DATA_BLOCK DB 17
TITLE =
{ S7_language := '7(1) Deutsch (Deutschland)  10.06.2014  10:57:37' }
AUTHOR : DAGO
FAMILY : PEPS
NAME : PEPS
VERSION : 0.1


  STRUCT
   alarms : STRUCT
    alarms : ARRAY  [1 .. 50 ] OF WORD;
   END_STRUCT ;
   LOT_DATA : STRUCT
    SON : STRING  [10 ];
    INR : STRING  [15 ];
    LOTSIZE : DINT ;
    SPARE_34 : DWORD ;
    SPARE_38 : DWORD ;
    SPARE_42 : DWORD ;
    SPARE_46 : DWORD ;
   END_STRUCT ;
   GENERAL : STRUCT
    MODE : INT ;
    RFD : BOOL ;
    RFU : BOOL ;
    RUN : BOOL ;
    IDLE : BOOL ;
    SPARE_2_4 : BOOL ;
    SPARE_2_5 : BOOL ;
    SPARE_2_6 : BOOL ;
    SPARE_2_7 : BOOL ;
    MACHINE_STARTED : BOOL ;	//Machine started
    AUTO : BOOL ;	//Auto visualisation
    MANUAL : BOOL ;	//Manual visualisation
    STELLEN : BOOL ;	//Stellen
    INFEED_BLOCKING : BOOL ;	//Infeed blocking visualisation
    PRODUCT_SUPPLY : BOOL ;	//Product supply visualisation
    PRE_PRODUCTION : BOOL ;	//Pr� production visualisation
    FILLING : BOOL ;	//Filling visualisation
    STOPPERS : BOOL  := TRUE;	//Stoppers visualisation
    IPC_SAMPLING : BOOL ;	//IPC sampling visualisation
    REJECT_ALL_SYRINGES : BOOL ;	//Reject all syringes visualisation
    RUN_EMPTY : BOOL ;	//Run empty machine visualisation
    START_UP : BOOL ;	//StartUp visualisation
    PRIMING : BOOL ;	//Priming visualisation
    PREPRODUCTION : BOOL ;	//Pr� production visualisation
    RECIRCULATION_DEACTIVE : BOOL ;	//Recirculation deactivated
    SPARE_5_0 : BOOL ;
    SPARE_5_1 : BOOL ;
    SPARE_5_2 : BOOL ;
    SPARE_5_3 : BOOL ;
    SPARE_5_4 : BOOL ;
    SPARE_5_5 : BOOL ;
    SPARE_5_6 : BOOL ;
    SPARE_5_7 : BOOL ;
    SPARE_6_0 : BOOL ;
    SPARE_6_1 : BOOL ;
    SPARE_6_2 : BOOL ;
    SPARE_6_3 : BOOL ;
    SPARE_6_4 : BOOL ;
    SPARE_6_5 : BOOL ;
    SPARE_6_6 : BOOL ;
    SPARE_6_7 : BOOL ;
    PHASE : INT ;	//Phase
    SUB_PHASE : INT ;	//Sub Phase
    SPARE_12 : INT ;
    SPARE_14 : INT ;
    SPARE_16 : INT ;
    SPARE_18 : INT ;
    SPARE_20 : INT ;
    SPARE_22 : INT ;
    SPARE_24 : INT ;
    SPARE_26 : INT ;
    SPARE_28 : INT ;
    SPARE_30 : INT ;
    SPARE_32 : INT ;
    SPARE_34 : INT ;
    SPARE_36 : INT ;
    SPARE_38 : INT ;
    SPARE_40 : INT ;
    SPARE_42 : INT ;
    SPARE_44 : INT ;
    SPARE_46 : INT ;
    SPARE_48 : WORD ;
   END_STRUCT ;
   COUNTERS : STRUCT
    TOTAL_GOOD : DINT ;	//Aantal goede stuks
    REJECT_FILLER_CAPPER : DINT ;	//Aantal uitgeworpen
    REJECT_PRIMING : INT ;	//Aantal gebruikt voor priming
    TOTAL_OBJECTS : DINT ;	//Totaal aantal
    FILLED_REJECTED : DINT ;	//Aantal gevuld en uitgeworpen
    NON_FILLED_REJECTED : DINT ;	//Aantal niet gevuld en uitgeworpen
    IPC_FILLED_SAMPLES : INT ;	//Aantal als staal genomen
    REJECT_NON_STARTUP : DINT ;	//Aantal fouten door geen opstart, priming of pr�-produktie uit te voeren
    SPARE_28 : INT ;
    REJECT_NEEDLE_DOWN : INT ;	//Aantal uitgeworpen na naalden uit positie
    REJECT_ALL_NON_FILL_SYR : DINT ;	//Aantal niet gevulde uitgeworpen door functie 'Alle syringes uitwerpen'
    REJECT_ALL_FILLED_SYR : DINT ;	//Aantal gevulde uitgeworpen door functie 'Alle syringes uitwerpen'
    FAULT_TIP_CAP_CONTR : INT ;	//Aantal fouten aan tip cap controlestation
    FAULT_TIP_CAP_CONTR_1 : INT ;	//Aantal fouten aan tip cap controle positie 1
    FAULT_TIP_CAP_CONTR_2 : INT ;	//Aantal fouten aan tip cap controle positie 2
    FAULT_TIP_CAP_CONTR_3 : INT ;	//Aantal fouten aan tip cap controle positie 3
    FAULT_TIP_CAP_CONTR_4 : INT ;	//Aantal fouten aan tip cap controle positie 4
    FAULT_STOPPER_CONTR : INT ;	//Aantal fouten aan stopper controlestation
    FAULT_STOPPER_CONTR_1 : INT ;	//Aantal fouten aan stopper controle positie 1
    FAULT_STOPPER_CONTR_2 : INT ;	//Aantal fouten aan stopper controle positie 2
    FAULT_STOPPER_CONTR_3 : INT ;	//Aantal fouten aan stopper controle positie 3
    FAULT_STOPPER_CONTR_4 : INT ;	//Aantal fouten aan stopper controle positie 4
    FAULT_STANDSTILL : DINT ;	//Aantal slecht door maximale stilstand overschreden
    FAULT_TUNNEL : DINT ;	//Aantal slecht door te lang in tunnel
    FAULT_ISOL_FILLED : DINT ;	//Aantal gevulde slecht door isolator
    FAULT_ISOL_NON_FILLED : DINT ;	//Aantal niet gevulde slecht door isolator
    FAULT_E_STOP_FILLED : DINT ;	//Aantal slechten onder vulnaalden door activatie noodstop
    FAULT_E_STOP_NON_FILLED : DINT ;	//Aantal slechten tussen vullen en stopperen door activatie noodstop
    REJECT_SMC_MODE : DINT ;	//Aantal uitgeworpen in SMC mode
    REJECT_JOG_MODE : DINT ;	//Aantal uitgeworpen in JOG mode
    SPARE_92 : DINT ;
    REJECT_RECIRCULATION : DINT ;	//Aantal uitgeworpen na recirculatie
    SPARE_100 : DINT ;
    SPARE_104 : DINT ;
    SPARE_108 : DINT ;
    SPARE_112 : DINT ;
    SPARE_116 : DINT ;
    SPARE_120 : DINT ;
    SPARE_124 : DINT ;
    SPARE_128 : INT ;
   END_STRUCT ;
   SPARE_288 : DWORD ;
   SPARE_292 : DWORD ;
   SPARE_296 : DWORD ;
   SPARE_290 : DWORD ;
   SPARE_294 : DWORD ;
  END_STRUCT ;
BEGIN
   ALARMS.ALARM[1] := FALSE;
   ALARMS.ALARM[2] := FALSE;
   ALARMS.ALARM[3] := FALSE;
   ALARMS.ALARM[4] := FALSE;
   ALARMS.ALARM[5] := FALSE;
   ALARMS.ALARM[6] := FALSE;
   ALARMS.ALARM[7] := FALSE;
   ALARMS.ALARM[8] := FALSE;
   ALARMS.ALARM[9] := FALSE;
   ALARMS.ALARM[10] := FALSE;
   ALARMS.ALARM[11] := FALSE;
   ALARMS.ALARM[12] := FALSE;
   ALARMS.ALARM[13] := FALSE;
   ALARMS.ALARM[14] := FALSE;
   ALARMS.ALARM[15] := FALSE;
   ALARMS.ALARM[16] := FALSE;
   ALARMS.ALARM[17] := FALSE;
   ALARMS.ALARM[18] := FALSE;
   ALARMS.ALARM[19] := FALSE;
   ALARMS.ALARM[20] := FALSE;
   ALARMS.ALARM[21] := FALSE;
   ALARMS.ALARM[22] := FALSE;
   ALARMS.ALARM[23] := FALSE;
   ALARMS.ALARM[24] := FALSE;
   ALARMS.ALARM[25] := FALSE;
   ALARMS.ALARM[26] := FALSE;
   ALARMS.ALARM[27] := FALSE;
   ALARMS.ALARM[28] := FALSE;
   ALARMS.ALARM[29] := FALSE;
   ALARMS.ALARM[30] := FALSE;
   ALARMS.ALARM[31] := FALSE;
   ALARMS.ALARM[32] := FALSE;
   ALARMS.ALARM[33] := FALSE;
   ALARMS.ALARM[34] := FALSE;
   ALARMS.ALARM[35] := FALSE;
   ALARMS.ALARM[36] := FALSE;
   ALARMS.ALARM[37] := FALSE;
   ALARMS.ALARM[38] := FALSE;
   ALARMS.ALARM[39] := FALSE;
   ALARMS.ALARM[40] := FALSE;
   ALARMS.ALARM[41] := FALSE;
   ALARMS.ALARM[42] := FALSE;
   ALARMS.ALARM[43] := FALSE;
   ALARMS.ALARM[44] := FALSE;
   ALARMS.ALARM[45] := FALSE;
   ALARMS.ALARM[46] := FALSE;
   ALARMS.ALARM[47] := FALSE;
   ALARMS.ALARM[48] := FALSE;
   ALARMS.ALARM[49] := FALSE;
   ALARMS.ALARM[50] := FALSE;
   ALARMS.ALARM[51] := FALSE;
   ALARMS.ALARM[52] := FALSE;
   ALARMS.ALARM[53] := FALSE;
   ALARMS.ALARM[54] := FALSE;
   ALARMS.ALARM[55] := FALSE;
   ALARMS.ALARM[56] := FALSE;
   ALARMS.ALARM[57] := FALSE;
   ALARMS.ALARM[58] := FALSE;
   ALARMS.ALARM[59] := FALSE;
   ALARMS.ALARM[60] := FALSE;
   ALARMS.ALARM[61] := FALSE;
   ALARMS.ALARM[62] := FALSE;
   ALARMS.ALARM[63] := FALSE;
   ALARMS.ALARM[64] := FALSE;
   ALARMS.ALARM[65] := FALSE;
   ALARMS.ALARM[66] := FALSE;
   ALARMS.ALARM[67] := FALSE;
   ALARMS.ALARM[68] := FALSE;
   ALARMS.ALARM[69] := FALSE;
   ALARMS.ALARM[70] := FALSE;
   ALARMS.ALARM[71] := FALSE;
   ALARMS.ALARM[72] := FALSE;
   ALARMS.ALARM[73] := FALSE;
   ALARMS.ALARM[74] := FALSE;
   ALARMS.ALARM[75] := FALSE;
   ALARMS.ALARM[76] := FALSE;
   ALARMS.ALARM[77] := FALSE;
   ALARMS.ALARM[78] := FALSE;
   ALARMS.ALARM[79] := FALSE;
   ALARMS.ALARM[80] := FALSE;
   ALARMS.ALARM[81] := FALSE;
   ALARMS.ALARM[82] := FALSE;
   ALARMS.ALARM[83] := FALSE;
   ALARMS.ALARM[84] := FALSE;
   ALARMS.ALARM[85] := FALSE;
   ALARMS.ALARM[86] := FALSE;
   ALARMS.ALARM[87] := FALSE;
   ALARMS.ALARM[88] := FALSE;
   ALARMS.ALARM[89] := FALSE;
   ALARMS.ALARM[90] := FALSE;
   ALARMS.ALARM[91] := FALSE;
   ALARMS.ALARM[92] := FALSE;
   ALARMS.ALARM[93] := FALSE;
   ALARMS.ALARM[94] := FALSE;
   ALARMS.ALARM[95] := FALSE;
   ALARMS.ALARM[96] := FALSE;
   ALARMS.ALARM[97] := FALSE;
   ALARMS.ALARM[98] := FALSE;
   ALARMS.ALARM[99] := FALSE;
   ALARMS.ALARM[100] := FALSE;
   ALARMS.ALARM[101] := FALSE;
   ALARMS.ALARM[102] := FALSE;
   ALARMS.ALARM[103] := FALSE;
   ALARMS.ALARM[104] := FALSE;
   ALARMS.ALARM[105] := FALSE;
   ALARMS.ALARM[106] := FALSE;
   ALARMS.ALARM[107] := FALSE;
   ALARMS.ALARM[108] := FALSE;
   ALARMS.ALARM[109] := FALSE;
   ALARMS.ALARM[110] := FALSE;
   ALARMS.ALARM[111] := FALSE;
   ALARMS.ALARM[112] := FALSE;
   ALARMS.ALARM[113] := FALSE;
   ALARMS.ALARM[114] := FALSE;
   ALARMS.ALARM[115] := FALSE;
   ALARMS.ALARM[116] := FALSE;
   ALARMS.ALARM[117] := FALSE;
   ALARMS.ALARM[118] := FALSE;
   ALARMS.ALARM[119] := FALSE;
   ALARMS.ALARM[120] := FALSE;
   ALARMS.ALARM[121] := FALSE;
   ALARMS.ALARM[122] := FALSE;
   ALARMS.ALARM[123] := FALSE;
   ALARMS.ALARM[124] := FALSE;
   ALARMS.ALARM[125] := FALSE;
   ALARMS.ALARM[126] := FALSE;
   ALARMS.ALARM[127] := FALSE;
   ALARMS.ALARM[128] := FALSE;
   ALARMS.ALARM[129] := FALSE;
   ALARMS.ALARM[130] := FALSE;
   ALARMS.ALARM[131] := FALSE;
   ALARMS.ALARM[132] := FALSE;
   ALARMS.ALARM[133] := FALSE;
   ALARMS.ALARM[134] := FALSE;
   ALARMS.ALARM[135] := FALSE;
   ALARMS.ALARM[136] := FALSE;
   ALARMS.ALARM[137] := FALSE;
   ALARMS.ALARM[138] := FALSE;
   ALARMS.ALARM[139] := FALSE;
   ALARMS.ALARM[140] := FALSE;
   ALARMS.ALARM[141] := FALSE;
   ALARMS.ALARM[142] := FALSE;
   ALARMS.ALARM[143] := FALSE;
   ALARMS.ALARM[144] := FALSE;
   ALARMS.ALARM[145] := FALSE;
   ALARMS.ALARM[146] := FALSE;
   ALARMS.ALARM[147] := FALSE;
   ALARMS.ALARM[148] := FALSE;
   ALARMS.ALARM[149] := FALSE;
   ALARMS.ALARM[150] := FALSE;
   ALARMS.ALARM[151] := FALSE;
   ALARMS.ALARM[152] := FALSE;
   ALARMS.ALARM[153] := FALSE;
   ALARMS.ALARM[154] := FALSE;
   ALARMS.ALARM[155] := FALSE;
   ALARMS.ALARM[156] := FALSE;
   ALARMS.ALARM[157] := FALSE;
   ALARMS.ALARM[158] := FALSE;
   ALARMS.ALARM[159] := FALSE;
   ALARMS.ALARM[160] := FALSE;
   ALARMS.ALARM[161] := FALSE;
   ALARMS.ALARM[162] := FALSE;
   ALARMS.ALARM[163] := FALSE;
   ALARMS.ALARM[164] := FALSE;
   ALARMS.ALARM[165] := FALSE;
   ALARMS.ALARM[166] := FALSE;
   ALARMS.ALARM[167] := FALSE;
   ALARMS.ALARM[168] := FALSE;
   ALARMS.ALARM[169] := FALSE;
   ALARMS.ALARM[170] := FALSE;
   ALARMS.ALARM[171] := FALSE;
   ALARMS.ALARM[172] := FALSE;
   ALARMS.ALARM[173] := FALSE;
   ALARMS.ALARM[174] := FALSE;
   ALARMS.ALARM[175] := FALSE;
   ALARMS.ALARM[176] := FALSE;
   ALARMS.ALARM[177] := FALSE;
   ALARMS.ALARM[178] := FALSE;
   ALARMS.ALARM[179] := FALSE;
   ALARMS.ALARM[180] := FALSE;
   ALARMS.ALARM[181] := FALSE;
   ALARMS.ALARM[182] := FALSE;
   ALARMS.ALARM[183] := FALSE;
   ALARMS.ALARM[184] := FALSE;
   ALARMS.ALARM[185] := FALSE;
   ALARMS.ALARM[186] := FALSE;
   ALARMS.ALARM[187] := FALSE;
   ALARMS.ALARM[188] := FALSE;
   ALARMS.ALARM[189] := FALSE;
   ALARMS.ALARM[190] := FALSE;
   ALARMS.ALARM[191] := FALSE;
   ALARMS.ALARM[192] := FALSE;
   ALARMS.ALARM[193] := FALSE;
   ALARMS.ALARM[194] := FALSE;
   ALARMS.ALARM[195] := FALSE;
   ALARMS.ALARM[196] := FALSE;
   ALARMS.ALARM[197] := FALSE;
   ALARMS.ALARM[198] := FALSE;
   ALARMS.ALARM[199] := FALSE;
   ALARMS.ALARM[200] := FALSE;
   ALARMS.ALARM[201] := FALSE;
   ALARMS.ALARM[202] := FALSE;
   ALARMS.ALARM[203] := FALSE;
   ALARMS.ALARM[204] := FALSE;
   ALARMS.ALARM[205] := FALSE;
   ALARMS.ALARM[206] := FALSE;
   ALARMS.ALARM[207] := FALSE;
   ALARMS.ALARM[208] := FALSE;
   ALARMS.ALARM[209] := FALSE;
   ALARMS.ALARM[210] := FALSE;
   ALARMS.ALARM[211] := FALSE;
   ALARMS.ALARM[212] := FALSE;
   ALARMS.ALARM[213] := FALSE;
   ALARMS.ALARM[214] := FALSE;
   ALARMS.ALARM[215] := FALSE;
   ALARMS.ALARM[216] := FALSE;
   ALARMS.ALARM[217] := FALSE;
   ALARMS.ALARM[218] := FALSE;
   ALARMS.ALARM[219] := FALSE;
   ALARMS.ALARM[220] := FALSE;
   ALARMS.ALARM[221] := FALSE;
   ALARMS.ALARM[222] := FALSE;
   ALARMS.ALARM[223] := FALSE;
   ALARMS.ALARM[224] := FALSE;
   ALARMS.ALARM[225] := FALSE;
   ALARMS.ALARM[226] := FALSE;
   ALARMS.ALARM[227] := FALSE;
   ALARMS.ALARM[228] := FALSE;
   ALARMS.ALARM[229] := FALSE;
   ALARMS.ALARM[230] := FALSE;
   ALARMS.ALARM[231] := FALSE;
   ALARMS.ALARM[232] := FALSE;
   ALARMS.ALARM[233] := FALSE;
   ALARMS.ALARM[234] := FALSE;
   ALARMS.ALARM[235] := FALSE;
   ALARMS.ALARM[236] := FALSE;
   ALARMS.ALARM[237] := FALSE;
   ALARMS.ALARM[238] := FALSE;
   ALARMS.ALARM[239] := FALSE;
   ALARMS.ALARM[240] := FALSE;
   ALARMS.ALARM[241] := FALSE;
   ALARMS.ALARM[242] := FALSE;
   ALARMS.ALARM[243] := FALSE;
   ALARMS.ALARM[244] := FALSE;
   ALARMS.ALARM[245] := FALSE;
   ALARMS.ALARM[246] := FALSE;
   ALARMS.ALARM[247] := FALSE;
   ALARMS.ALARM[248] := FALSE;
   ALARMS.ALARM[249] := FALSE;
   ALARMS.ALARM[250] := FALSE;
   ALARMS.ALARM[251] := FALSE;
   ALARMS.ALARM[252] := FALSE;
   ALARMS.ALARM[253] := FALSE;
   ALARMS.ALARM[254] := FALSE;
   ALARMS.ALARM[255] := FALSE;
   ALARMS.ALARM[256] := FALSE;
   ALARMS.ALARM[257] := FALSE;
   ALARMS.ALARM[258] := FALSE;
   ALARMS.ALARM[259] := FALSE;
   ALARMS.ALARM[260] := FALSE;
   ALARMS.ALARM[261] := FALSE;
   ALARMS.ALARM[262] := FALSE;
   ALARMS.ALARM[263] := FALSE;
   ALARMS.ALARM[264] := FALSE;
   ALARMS.ALARM[265] := FALSE;
   ALARMS.ALARM[266] := FALSE;
   ALARMS.ALARM[267] := FALSE;
   ALARMS.ALARM[268] := FALSE;
   ALARMS.ALARM[269] := FALSE;
   ALARMS.ALARM[270] := FALSE;
   ALARMS.ALARM[271] := FALSE;
   ALARMS.ALARM[272] := FALSE;
   ALARMS.ALARM[273] := FALSE;
   ALARMS.ALARM[274] := FALSE;
   ALARMS.ALARM[275] := FALSE;
   ALARMS.ALARM[276] := FALSE;
   ALARMS.ALARM[277] := FALSE;
   ALARMS.ALARM[278] := FALSE;
   ALARMS.ALARM[279] := FALSE;
   ALARMS.ALARM[280] := FALSE;
   ALARMS.ALARM[281] := FALSE;
   ALARMS.ALARM[282] := FALSE;
   ALARMS.ALARM[283] := FALSE;
   ALARMS.ALARM[284] := FALSE;
   ALARMS.ALARM[285] := FALSE;
   ALARMS.ALARM[286] := FALSE;
   ALARMS.ALARM[287] := FALSE;
   ALARMS.ALARM[288] := FALSE;
   ALARMS.ALARM[289] := FALSE;
   ALARMS.ALARM[290] := FALSE;
   ALARMS.ALARM[291] := FALSE;
   ALARMS.ALARM[292] := FALSE;
   ALARMS.ALARM[293] := FALSE;
   ALARMS.ALARM[294] := FALSE;
   ALARMS.ALARM[295] := FALSE;
   ALARMS.ALARM[296] := FALSE;
   ALARMS.ALARM[297] := FALSE;
   ALARMS.ALARM[298] := FALSE;
   ALARMS.ALARM[299] := FALSE;
   ALARMS.ALARM[300] := FALSE;
   ALARMS.ALARM[301] := FALSE;
   ALARMS.ALARM[302] := FALSE;
   ALARMS.ALARM[303] := FALSE;
   ALARMS.ALARM[304] := FALSE;
   ALARMS.ALARM[305] := FALSE;
   ALARMS.ALARM[306] := FALSE;
   ALARMS.ALARM[307] := FALSE;
   ALARMS.ALARM[308] := FALSE;
   ALARMS.ALARM[309] := FALSE;
   ALARMS.ALARM[310] := FALSE;
   ALARMS.ALARM[311] := FALSE;
   ALARMS.ALARM[312] := FALSE;
   ALARMS.ALARM[313] := FALSE;
   ALARMS.ALARM[314] := FALSE;
   ALARMS.ALARM[315] := FALSE;
   ALARMS.ALARM[316] := FALSE;
   ALARMS.ALARM[317] := FALSE;
   ALARMS.ALARM[318] := FALSE;
   ALARMS.ALARM[319] := FALSE;
   ALARMS.ALARM[320] := FALSE;
   ALARMS.ALARM[321] := FALSE;
   ALARMS.ALARM[322] := FALSE;
   ALARMS.ALARM[323] := FALSE;
   ALARMS.ALARM[324] := FALSE;
   ALARMS.ALARM[325] := FALSE;
   ALARMS.ALARM[326] := FALSE;
   ALARMS.ALARM[327] := FALSE;
   ALARMS.ALARM[328] := FALSE;
   ALARMS.ALARM[329] := FALSE;
   ALARMS.ALARM[330] := FALSE;
   ALARMS.ALARM[331] := FALSE;
   ALARMS.ALARM[332] := FALSE;
   ALARMS.ALARM[333] := FALSE;
   ALARMS.ALARM[334] := FALSE;
   ALARMS.ALARM[335] := FALSE;
   ALARMS.ALARM[336] := FALSE;
   ALARMS.ALARM[337] := FALSE;
   ALARMS.ALARM[338] := FALSE;
   ALARMS.ALARM[339] := FALSE;
   ALARMS.ALARM[340] := FALSE;
   ALARMS.ALARM[341] := FALSE;
   ALARMS.ALARM[342] := FALSE;
   ALARMS.ALARM[343] := FALSE;
   ALARMS.ALARM[344] := FALSE;
   ALARMS.ALARM[345] := FALSE;
   ALARMS.ALARM[346] := FALSE;
   ALARMS.ALARM[347] := FALSE;
   ALARMS.ALARM[348] := FALSE;
   ALARMS.ALARM[349] := FALSE;
   ALARMS.ALARM[350] := FALSE;
   ALARMS.ALARM[351] := FALSE;
   ALARMS.ALARM[352] := FALSE;
   ALARMS.ALARM[353] := FALSE;
   ALARMS.ALARM[354] := FALSE;
   ALARMS.ALARM[355] := FALSE;
   ALARMS.ALARM[356] := FALSE;
   ALARMS.ALARM[357] := FALSE;
   ALARMS.ALARM[358] := FALSE;
   ALARMS.ALARM[359] := FALSE;
   ALARMS.ALARM[360] := FALSE;
   ALARMS.ALARM[361] := FALSE;
   ALARMS.ALARM[362] := FALSE;
   ALARMS.ALARM[363] := FALSE;
   ALARMS.ALARM[364] := FALSE;
   ALARMS.ALARM[365] := FALSE;
   ALARMS.ALARM[366] := FALSE;
   ALARMS.ALARM[367] := FALSE;
   ALARMS.ALARM[368] := FALSE;
   ALARMS.ALARM[369] := FALSE;
   ALARMS.ALARM[370] := FALSE;
   ALARMS.ALARM[371] := FALSE;
   ALARMS.ALARM[372] := FALSE;
   ALARMS.ALARM[373] := FALSE;
   ALARMS.ALARM[374] := FALSE;
   ALARMS.ALARM[375] := FALSE;
   ALARMS.ALARM[376] := FALSE;
   ALARMS.ALARM[377] := FALSE;
   ALARMS.ALARM[378] := FALSE;
   ALARMS.ALARM[379] := FALSE;
   ALARMS.ALARM[380] := FALSE;
   ALARMS.ALARM[381] := FALSE;
   ALARMS.ALARM[382] := FALSE;
   ALARMS.ALARM[383] := FALSE;
   ALARMS.ALARM[384] := FALSE;
   ALARMS.ALARM[385] := FALSE;
   ALARMS.ALARM[386] := FALSE;
   ALARMS.ALARM[387] := FALSE;
   ALARMS.ALARM[388] := FALSE;
   ALARMS.ALARM[389] := FALSE;
   ALARMS.ALARM[390] := FALSE;
   ALARMS.ALARM[391] := FALSE;
   ALARMS.ALARM[392] := FALSE;
   ALARMS.ALARM[393] := FALSE;
   ALARMS.ALARM[394] := FALSE;
   ALARMS.ALARM[395] := FALSE;
   ALARMS.ALARM[396] := FALSE;
   ALARMS.ALARM[397] := FALSE;
   ALARMS.ALARM[398] := FALSE;
   ALARMS.ALARM[399] := FALSE;
   ALARMS.ALARM[400] := FALSE;
   ALARMS.ALARM[401] := FALSE;
   ALARMS.ALARM[402] := FALSE;
   ALARMS.ALARM[403] := FALSE;
   ALARMS.ALARM[404] := FALSE;
   ALARMS.ALARM[405] := FALSE;
   ALARMS.ALARM[406] := FALSE;
   ALARMS.ALARM[407] := FALSE;
   ALARMS.ALARM[408] := FALSE;
   ALARMS.ALARM[409] := FALSE;
   ALARMS.ALARM[410] := FALSE;
   ALARMS.ALARM[411] := FALSE;
   ALARMS.ALARM[412] := FALSE;
   ALARMS.ALARM[413] := FALSE;
   ALARMS.ALARM[414] := FALSE;
   ALARMS.ALARM[415] := FALSE;
   ALARMS.ALARM[416] := FALSE;
   ALARMS.ALARM[417] := FALSE;
   ALARMS.ALARM[418] := FALSE;
   ALARMS.ALARM[419] := FALSE;
   ALARMS.ALARM[420] := FALSE;
   ALARMS.ALARM[421] := FALSE;
   ALARMS.ALARM[422] := FALSE;
   ALARMS.ALARM[423] := FALSE;
   ALARMS.ALARM[424] := FALSE;
   ALARMS.ALARM[425] := FALSE;
   ALARMS.ALARM[426] := FALSE;
   ALARMS.ALARM[427] := FALSE;
   ALARMS.ALARM[428] := FALSE;
   ALARMS.ALARM[429] := FALSE;
   ALARMS.ALARM[430] := FALSE;
   ALARMS.ALARM[431] := FALSE;
   ALARMS.ALARM[432] := FALSE;
   ALARMS.ALARM[433] := FALSE;
   ALARMS.ALARM[434] := FALSE;
   ALARMS.ALARM[435] := FALSE;
   ALARMS.ALARM[436] := FALSE;
   ALARMS.ALARM[437] := FALSE;
   ALARMS.ALARM[438] := FALSE;
   ALARMS.ALARM[439] := FALSE;
   ALARMS.ALARM[440] := FALSE;
   ALARMS.ALARM[441] := FALSE;
   ALARMS.ALARM[442] := FALSE;
   ALARMS.ALARM[443] := FALSE;
   ALARMS.ALARM[444] := FALSE;
   ALARMS.ALARM[445] := FALSE;
   ALARMS.ALARM[446] := FALSE;
   ALARMS.ALARM[447] := FALSE;
   ALARMS.ALARM[448] := FALSE;
   ALARMS.ALARM[449] := FALSE;
   ALARMS.ALARM[450] := FALSE;
   ALARMS.ALARM[451] := FALSE;
   ALARMS.ALARM[452] := FALSE;
   ALARMS.ALARM[453] := FALSE;
   ALARMS.ALARM[454] := FALSE;
   ALARMS.ALARM[455] := FALSE;
   ALARMS.ALARM[456] := FALSE;
   ALARMS.ALARM[457] := FALSE;
   ALARMS.ALARM[458] := FALSE;
   ALARMS.ALARM[459] := FALSE;
   ALARMS.ALARM[460] := FALSE;
   ALARMS.ALARM[461] := FALSE;
   ALARMS.ALARM[462] := FALSE;
   ALARMS.ALARM[463] := FALSE;
   ALARMS.ALARM[464] := FALSE;
   ALARMS.ALARM[465] := FALSE;
   ALARMS.ALARM[466] := FALSE;
   ALARMS.ALARM[467] := FALSE;
   ALARMS.ALARM[468] := FALSE;
   ALARMS.ALARM[469] := FALSE;
   ALARMS.ALARM[470] := FALSE;
   ALARMS.ALARM[471] := FALSE;
   ALARMS.ALARM[472] := FALSE;
   ALARMS.ALARM[473] := FALSE;
   ALARMS.ALARM[474] := FALSE;
   ALARMS.ALARM[475] := FALSE;
   ALARMS.ALARM[476] := FALSE;
   ALARMS.ALARM[477] := FALSE;
   ALARMS.ALARM[478] := FALSE;
   ALARMS.ALARM[479] := FALSE;
   ALARMS.ALARM[480] := FALSE;
   ALARMS.ALARM[481] := FALSE;
   ALARMS.ALARM[482] := FALSE;
   ALARMS.ALARM[483] := FALSE;
   ALARMS.ALARM[484] := FALSE;
   ALARMS.ALARM[485] := FALSE;
   ALARMS.ALARM[486] := FALSE;
   ALARMS.ALARM[487] := FALSE;
   ALARMS.ALARM[488] := FALSE;
   ALARMS.ALARM[489] := FALSE;
   ALARMS.ALARM[490] := FALSE;
   ALARMS.ALARM[491] := FALSE;
   ALARMS.ALARM[492] := FALSE;
   ALARMS.ALARM[493] := FALSE;
   ALARMS.ALARM[494] := FALSE;
   ALARMS.ALARM[495] := FALSE;
   ALARMS.ALARM[496] := FALSE;
   ALARMS.ALARM[497] := FALSE;
   ALARMS.ALARM[498] := FALSE;
   ALARMS.ALARM[499] := FALSE;
   ALARMS.ALARM[500] := FALSE;
   ALARMS.ALARM[501] := FALSE;
   ALARMS.ALARM[502] := FALSE;
   ALARMS.ALARM[503] := FALSE;
   ALARMS.ALARM[504] := FALSE;
   ALARMS.ALARM[505] := FALSE;
   ALARMS.ALARM[506] := FALSE;
   ALARMS.ALARM[507] := FALSE;
   ALARMS.ALARM[508] := FALSE;
   ALARMS.ALARM[509] := FALSE;
   ALARMS.ALARM[510] := FALSE;
   ALARMS.ALARM[511] := FALSE;
   ALARMS.ALARM[512] := FALSE;
   ALARMS.ALARM[513] := FALSE;
   ALARMS.ALARM[514] := FALSE;
   ALARMS.ALARM[515] := FALSE;
   ALARMS.ALARM[516] := FALSE;
   ALARMS.ALARM[517] := FALSE;
   ALARMS.ALARM[518] := FALSE;
   ALARMS.ALARM[519] := FALSE;
   ALARMS.ALARM[520] := FALSE;
   ALARMS.ALARM[521] := FALSE;
   ALARMS.ALARM[522] := FALSE;
   ALARMS.ALARM[523] := FALSE;
   ALARMS.ALARM[524] := FALSE;
   ALARMS.ALARM[525] := FALSE;
   ALARMS.ALARM[526] := FALSE;
   ALARMS.ALARM[527] := FALSE;
   ALARMS.ALARM[528] := FALSE;
   ALARMS.ALARM[529] := FALSE;
   ALARMS.ALARM[530] := FALSE;
   ALARMS.ALARM[531] := FALSE;
   ALARMS.ALARM[532] := FALSE;
   ALARMS.ALARM[533] := FALSE;
   ALARMS.ALARM[534] := FALSE;
   ALARMS.ALARM[535] := FALSE;
   ALARMS.ALARM[536] := FALSE;
   ALARMS.ALARM[537] := FALSE;
   ALARMS.ALARM[538] := FALSE;
   ALARMS.ALARM[539] := FALSE;
   ALARMS.ALARM[540] := FALSE;
   ALARMS.ALARM[541] := FALSE;
   ALARMS.ALARM[542] := FALSE;
   ALARMS.ALARM[543] := FALSE;
   ALARMS.ALARM[544] := FALSE;
   ALARMS.ALARM[545] := FALSE;
   ALARMS.ALARM[546] := FALSE;
   ALARMS.ALARM[547] := FALSE;
   ALARMS.ALARM[548] := FALSE;
   ALARMS.ALARM[549] := FALSE;
   ALARMS.ALARM[550] := FALSE;
   ALARMS.ALARM[551] := FALSE;
   ALARMS.ALARM[552] := FALSE;
   ALARMS.ALARM[553] := FALSE;
   ALARMS.ALARM[554] := FALSE;
   ALARMS.ALARM[555] := FALSE;
   ALARMS.ALARM[556] := FALSE;
   ALARMS.ALARM[557] := FALSE;
   ALARMS.ALARM[558] := FALSE;
   ALARMS.ALARM[559] := FALSE;
   ALARMS.ALARM[560] := FALSE;
   ALARMS.ALARM[561] := FALSE;
   ALARMS.ALARM[562] := FALSE;
   ALARMS.ALARM[563] := FALSE;
   ALARMS.ALARM[564] := FALSE;
   ALARMS.ALARM[565] := FALSE;
   ALARMS.ALARM[566] := FALSE;
   ALARMS.ALARM[567] := FALSE;
   ALARMS.ALARM[568] := FALSE;
   ALARMS.ALARM[569] := FALSE;
   ALARMS.ALARM[570] := FALSE;
   ALARMS.ALARM[571] := FALSE;
   ALARMS.ALARM[572] := FALSE;
   ALARMS.ALARM[573] := FALSE;
   ALARMS.ALARM[574] := FALSE;
   ALARMS.ALARM[575] := FALSE;
   ALARMS.ALARM[576] := FALSE;
   ALARMS.ALARM[577] := FALSE;
   ALARMS.ALARM[578] := FALSE;
   ALARMS.ALARM[579] := FALSE;
   ALARMS.ALARM[580] := FALSE;
   ALARMS.ALARM[581] := FALSE;
   ALARMS.ALARM[582] := FALSE;
   ALARMS.ALARM[583] := FALSE;
   ALARMS.ALARM[584] := FALSE;
   ALARMS.ALARM[585] := FALSE;
   ALARMS.ALARM[586] := FALSE;
   ALARMS.ALARM[587] := FALSE;
   ALARMS.ALARM[588] := FALSE;
   ALARMS.ALARM[589] := FALSE;
   ALARMS.ALARM[590] := FALSE;
   ALARMS.ALARM[591] := FALSE;
   ALARMS.ALARM[592] := FALSE;
   ALARMS.ALARM[593] := FALSE;
   ALARMS.ALARM[594] := FALSE;
   ALARMS.ALARM[595] := FALSE;
   ALARMS.ALARM[596] := FALSE;
   ALARMS.ALARM[597] := FALSE;
   ALARMS.ALARM[598] := FALSE;
   ALARMS.ALARM[599] := FALSE;
   ALARMS.ALARM[600] := FALSE;
   ALARMS.ALARM[601] := FALSE;
   ALARMS.ALARM[602] := FALSE;
   ALARMS.ALARM[603] := FALSE;
   ALARMS.ALARM[604] := FALSE;
   ALARMS.ALARM[605] := FALSE;
   ALARMS.ALARM[606] := FALSE;
   ALARMS.ALARM[607] := FALSE;
   ALARMS.ALARM[608] := FALSE;
   ALARMS.ALARM[609] := FALSE;
   ALARMS.ALARM[610] := FALSE;
   ALARMS.ALARM[611] := FALSE;
   ALARMS.ALARM[612] := FALSE;
   ALARMS.ALARM[613] := FALSE;
   ALARMS.ALARM[614] := FALSE;
   ALARMS.ALARM[615] := FALSE;
   ALARMS.ALARM[616] := FALSE;
   ALARMS.ALARM[617] := FALSE;
   ALARMS.ALARM[618] := FALSE;
   ALARMS.ALARM[619] := FALSE;
   ALARMS.ALARM[620] := FALSE;
   ALARMS.ALARM[621] := FALSE;
   ALARMS.ALARM[622] := FALSE;
   ALARMS.ALARM[623] := FALSE;
   ALARMS.ALARM[624] := FALSE;
   ALARMS.ALARM[625] := FALSE;
   ALARMS.ALARM[626] := FALSE;
   ALARMS.ALARM[627] := FALSE;
   ALARMS.ALARM[628] := FALSE;
   ALARMS.ALARM[629] := FALSE;
   ALARMS.ALARM[630] := FALSE;
   ALARMS.ALARM[631] := FALSE;
   ALARMS.ALARM[632] := FALSE;
   ALARMS.ALARM[633] := FALSE;
   ALARMS.ALARM[634] := FALSE;
   ALARMS.ALARM[635] := FALSE;
   ALARMS.ALARM[636] := FALSE;
   ALARMS.ALARM[637] := FALSE;
   ALARMS.ALARM[638] := FALSE;
   ALARMS.ALARM[639] := FALSE;
   ALARMS.ALARM[640] := FALSE;
   ALARMS.ALARM[641] := FALSE;
   ALARMS.ALARM[642] := FALSE;
   ALARMS.ALARM[643] := FALSE;
   ALARMS.ALARM[644] := FALSE;
   ALARMS.ALARM[645] := FALSE;
   ALARMS.ALARM[646] := FALSE;
   ALARMS.ALARM[647] := FALSE;
   ALARMS.ALARM[648] := FALSE;
   ALARMS.ALARM[649] := FALSE;
   ALARMS.ALARM[650] := FALSE;
   ALARMS.ALARM[651] := FALSE;
   ALARMS.ALARM[652] := FALSE;
   ALARMS.ALARM[653] := FALSE;
   ALARMS.ALARM[654] := FALSE;
   ALARMS.ALARM[655] := FALSE;
   ALARMS.ALARM[656] := FALSE;
   ALARMS.ALARM[657] := FALSE;
   ALARMS.ALARM[658] := FALSE;
   ALARMS.ALARM[659] := FALSE;
   ALARMS.ALARM[660] := FALSE;
   ALARMS.ALARM[661] := FALSE;
   ALARMS.ALARM[662] := FALSE;
   ALARMS.ALARM[663] := FALSE;
   ALARMS.ALARM[664] := FALSE;
   ALARMS.ALARM[665] := FALSE;
   ALARMS.ALARM[666] := FALSE;
   ALARMS.ALARM[667] := FALSE;
   ALARMS.ALARM[668] := FALSE;
   ALARMS.ALARM[669] := FALSE;
   ALARMS.ALARM[670] := FALSE;
   ALARMS.ALARM[671] := FALSE;
   ALARMS.ALARM[672] := FALSE;
   ALARMS.ALARM[673] := FALSE;
   ALARMS.ALARM[674] := FALSE;
   ALARMS.ALARM[675] := FALSE;
   ALARMS.ALARM[676] := FALSE;
   ALARMS.ALARM[677] := FALSE;
   ALARMS.ALARM[678] := FALSE;
   ALARMS.ALARM[679] := FALSE;
   ALARMS.ALARM[680] := FALSE;
   ALARMS.ALARM[681] := FALSE;
   ALARMS.ALARM[682] := FALSE;
   ALARMS.ALARM[683] := FALSE;
   ALARMS.ALARM[684] := FALSE;
   ALARMS.ALARM[685] := FALSE;
   ALARMS.ALARM[686] := FALSE;
   ALARMS.ALARM[687] := FALSE;
   ALARMS.ALARM[688] := FALSE;
   ALARMS.ALARM[689] := FALSE;
   ALARMS.ALARM[690] := FALSE;
   ALARMS.ALARM[691] := FALSE;
   ALARMS.ALARM[692] := FALSE;
   ALARMS.ALARM[693] := FALSE;
   ALARMS.ALARM[694] := FALSE;
   ALARMS.ALARM[695] := FALSE;
   ALARMS.ALARM[696] := FALSE;
   ALARMS.ALARM[697] := FALSE;
   ALARMS.ALARM[698] := FALSE;
   ALARMS.ALARM[699] := FALSE;
   ALARMS.ALARM[700] := FALSE;
   ALARMS.ALARM[701] := FALSE;
   ALARMS.ALARM[702] := FALSE;
   ALARMS.ALARM[703] := FALSE;
   ALARMS.ALARM[704] := FALSE;
   ALARMS.ALARM[705] := FALSE;
   ALARMS.ALARM[706] := FALSE;
   ALARMS.ALARM[707] := FALSE;
   ALARMS.ALARM[708] := FALSE;
   ALARMS.ALARM[709] := FALSE;
   ALARMS.ALARM[710] := FALSE;
   ALARMS.ALARM[711] := FALSE;
   ALARMS.ALARM[712] := FALSE;
   ALARMS.ALARM[713] := FALSE;
   ALARMS.ALARM[714] := FALSE;
   ALARMS.ALARM[715] := FALSE;
   ALARMS.ALARM[716] := FALSE;
   ALARMS.ALARM[717] := FALSE;
   ALARMS.ALARM[718] := FALSE;
   ALARMS.ALARM[719] := FALSE;
   ALARMS.ALARM[720] := FALSE;
   ALARMS.ALARM[721] := FALSE;
   ALARMS.ALARM[722] := FALSE;
   ALARMS.ALARM[723] := FALSE;
   ALARMS.ALARM[724] := FALSE;
   ALARMS.ALARM[725] := FALSE;
   ALARMS.ALARM[726] := FALSE;
   ALARMS.ALARM[727] := FALSE;
   ALARMS.ALARM[728] := FALSE;
   ALARMS.ALARM[729] := FALSE;
   ALARMS.ALARM[730] := FALSE;
   ALARMS.ALARM[731] := FALSE;
   ALARMS.ALARM[732] := FALSE;
   ALARMS.ALARM[733] := FALSE;
   ALARMS.ALARM[734] := FALSE;
   ALARMS.ALARM[735] := FALSE;
   ALARMS.ALARM[736] := FALSE;
   ALARMS.ALARM[737] := FALSE;
   ALARMS.ALARM[738] := FALSE;
   ALARMS.ALARM[739] := FALSE;
   ALARMS.ALARM[740] := FALSE;
   ALARMS.ALARM[741] := FALSE;
   ALARMS.ALARM[742] := FALSE;
   ALARMS.ALARM[743] := FALSE;
   ALARMS.ALARM[744] := FALSE;
   ALARMS.ALARM[745] := FALSE;
   ALARMS.ALARM[746] := FALSE;
   ALARMS.ALARM[747] := FALSE;
   ALARMS.ALARM[748] := FALSE;
   ALARMS.ALARM[749] := FALSE;
   ALARMS.ALARM[750] := FALSE;
   ALARMS.ALARM[751] := FALSE;
   ALARMS.ALARM[752] := FALSE;
   ALARMS.ALARM[753] := FALSE;
   ALARMS.ALARM[754] := FALSE;
   ALARMS.ALARM[755] := FALSE;
   ALARMS.ALARM[756] := FALSE;
   ALARMS.ALARM[757] := FALSE;
   ALARMS.ALARM[758] := FALSE;
   ALARMS.ALARM[759] := FALSE;
   ALARMS.ALARM[760] := FALSE;
   ALARMS.ALARM[761] := FALSE;
   ALARMS.ALARM[762] := FALSE;
   ALARMS.ALARM[763] := FALSE;
   ALARMS.ALARM[764] := FALSE;
   ALARMS.ALARM[765] := FALSE;
   ALARMS.ALARM[766] := FALSE;
   ALARMS.ALARM[767] := FALSE;
   ALARMS.ALARM[768] := FALSE;
   ALARMS.ALARM[769] := FALSE;
   ALARMS.ALARM[770] := FALSE;
   ALARMS.ALARM[771] := FALSE;
   ALARMS.ALARM[772] := FALSE;
   ALARMS.ALARM[773] := FALSE;
   ALARMS.ALARM[774] := FALSE;
   ALARMS.ALARM[775] := FALSE;
   ALARMS.ALARM[776] := FALSE;
   ALARMS.ALARM[777] := FALSE;
   ALARMS.ALARM[778] := FALSE;
   ALARMS.ALARM[779] := FALSE;
   ALARMS.ALARM[780] := FALSE;
   ALARMS.ALARM[781] := FALSE;
   ALARMS.ALARM[782] := FALSE;
   ALARMS.ALARM[783] := FALSE;
   ALARMS.ALARM[784] := FALSE;
   ALARMS.ALARM[785] := FALSE;
   ALARMS.ALARM[786] := FALSE;
   ALARMS.ALARM[787] := FALSE;
   ALARMS.ALARM[788] := FALSE;
   ALARMS.ALARM[789] := FALSE;
   ALARMS.ALARM[790] := FALSE;
   ALARMS.ALARM[791] := FALSE;
   ALARMS.ALARM[792] := FALSE;
   ALARMS.ALARM[793] := FALSE;
   ALARMS.ALARM[794] := FALSE;
   ALARMS.ALARM[795] := FALSE;
   ALARMS.ALARM[796] := FALSE;
   ALARMS.ALARM[797] := FALSE;
   ALARMS.ALARM[798] := FALSE;
   ALARMS.ALARM[799] := FALSE;
   ALARMS.ALARM[800] := FALSE;
   LOT_DATA.SON := '';
   LOT_DATA.INR := '';
   LOT_DATA.LOTSIZE := L#0;
   LOT_DATA.SPARE_34 := DW#16#0;
   LOT_DATA.SPARE_38 := DW#16#0;
   LOT_DATA.SPARE_42 := DW#16#0;
   LOT_DATA.SPARE_46 := DW#16#0;
   GENERAL.MODE := 0;
   GENERAL.RFD := FALSE;
   GENERAL.RFU := FALSE;
   GENERAL.RUN := FALSE;
   GENERAL.IDLE := FALSE;
   GENERAL.SPARE_2_4 := FALSE;
   GENERAL.SPARE_2_5 := FALSE;
   GENERAL.SPARE_2_6 := FALSE;
   GENERAL.SPARE_2_7 := FALSE;
   GENERAL.MACHINE_STARTED := FALSE;
   GENERAL.AUTO := FALSE;
   GENERAL.MANUAL := FALSE;
   GENERAL.STELLEN := FALSE;
   GENERAL.INFEED_BLOCKING := FALSE;
   GENERAL.PRODUCT_SUPPLY := FALSE;
   GENERAL.PRE_PRODUCTION := FALSE;
   GENERAL.FILLING := FALSE;
   GENERAL.STOPPERS := TRUE;
   GENERAL.IPC_SAMPLING := FALSE;
   GENERAL.REJECT_ALL_SYRINGES := FALSE;
   GENERAL.RUN_EMPTY := FALSE;
   GENERAL.START_UP := FALSE;
   GENERAL.PRIMING := FALSE;
   GENERAL.PREPRODUCTION := FALSE;
   GENERAL.RECIRCULATION_DEACTIVE := FALSE;
   GENERAL.SPARE_5_0 := FALSE;
   GENERAL.SPARE_5_1 := FALSE;
   GENERAL.SPARE_5_2 := FALSE;
   GENERAL.SPARE_5_3 := FALSE;
   GENERAL.SPARE_5_4 := FALSE;
   GENERAL.SPARE_5_5 := FALSE;
   GENERAL.SPARE_5_6 := FALSE;
   GENERAL.SPARE_5_7 := FALSE;
   GENERAL.SPARE_6_0 := FALSE;
   GENERAL.SPARE_6_1 := FALSE;
   GENERAL.SPARE_6_2 := FALSE;
   GENERAL.SPARE_6_3 := FALSE;
   GENERAL.SPARE_6_4 := FALSE;
   GENERAL.SPARE_6_5 := FALSE;
   GENERAL.SPARE_6_6 := FALSE;
   GENERAL.SPARE_6_7 := FALSE;
   GENERAL.PHASE := 0;
   GENERAL.SUB_PHASE := 0;
   GENERAL.SPARE_12 := 0;
   GENERAL.SPARE_14 := 0;
   GENERAL.SPARE_16 := 0;
   GENERAL.SPARE_18 := 0;
   GENERAL.SPARE_20 := 0;
   GENERAL.SPARE_22 := 0;
   GENERAL.SPARE_24 := 0;
   GENERAL.SPARE_26 := 0;
   GENERAL.SPARE_28 := 0;
   GENERAL.SPARE_30 := 0;
   GENERAL.SPARE_32 := 0;
   GENERAL.SPARE_34 := 0;
   GENERAL.SPARE_36 := 0;
   GENERAL.SPARE_38 := 0;
   GENERAL.SPARE_40 := 0;
   GENERAL.SPARE_42 := 0;
   GENERAL.SPARE_44 := 0;
   GENERAL.SPARE_46 := 0;
   GENERAL.SPARE_48 := W#16#0;
   COUNTERS.TOTAL_GOOD := L#0;
   COUNTERS.REJECT_FILLER_CAPPER := L#0;
   COUNTERS.REJECT_PRIMING := 0;
   COUNTERS.TOTAL_OBJECTS := L#0;
   COUNTERS.FILLED_REJECTED := L#0;
   COUNTERS.NON_FILLED_REJECTED := L#0;
   COUNTERS.IPC_FILLED_SAMPLES := 0;
   COUNTERS.REJECT_NON_STARTUP := L#0;
   COUNTERS.SPARE_28 := 0;
   COUNTERS.REJECT_NEEDLE_DOWN := 0;
   COUNTERS.REJECT_ALL_NON_FILL_SYR := L#0;
   COUNTERS.REJECT_ALL_FILLED_SYR := L#0;
   COUNTERS.FAULT_TIP_CAP_CONTR := 0;
   COUNTERS.FAULT_TIP_CAP_CONTR_1 := 0;
   COUNTERS.FAULT_TIP_CAP_CONTR_2 := 0;
   COUNTERS.FAULT_TIP_CAP_CONTR_3 := 0;
   COUNTERS.FAULT_TIP_CAP_CONTR_4 := 0;
   COUNTERS.FAULT_STOPPER_CONTR := 0;
   COUNTERS.FAULT_STOPPER_CONTR_1 := 0;
   COUNTERS.FAULT_STOPPER_CONTR_2 := 0;
   COUNTERS.FAULT_STOPPER_CONTR_3 := 0;
   COUNTERS.FAULT_STOPPER_CONTR_4 := 0;
   COUNTERS.FAULT_STANDSTILL := L#0;
   COUNTERS.FAULT_TUNNEL := L#0;
   COUNTERS.FAULT_ISOL_FILLED := L#0;
   COUNTERS.FAULT_ISOL_NON_FILLED := L#0;
   COUNTERS.FAULT_E_STOP_FILLED := L#0;
   COUNTERS.FAULT_E_STOP_NON_FILLED := L#0;
   COUNTERS.REJECT_SMC_MODE := L#0;
   COUNTERS.REJECT_JOG_MODE := L#0;
   COUNTERS.SPARE_92 := L#0;
   COUNTERS.REJECT_RECIRCULATION := L#0;
   COUNTERS.SPARE_100 := L#0;
   COUNTERS.SPARE_104 := L#0;
   COUNTERS.SPARE_108 := L#0;
   COUNTERS.SPARE_112 := L#0;
   COUNTERS.SPARE_116 := L#0;
   COUNTERS.SPARE_120 := L#0;
   COUNTERS.SPARE_124 := L#0;
   COUNTERS.SPARE_128 := 0;
   SPARE_288 := DW#16#0;
   SPARE_292 := DW#16#0;
   SPARE_296 := DW#16#0;
   SPARE_290 := DW#16#0;
   SPARE_294 := DW#16#0;
END_DATA_BLOCK

